FUNCTION_BLOCK LedLamp
VAR_INPUT
END_VAR
VAR_OUTPUT
END_VAR
VAR
	output AT %Q* : BOOL;
END_VAR

PROPERTY IsOff : BOOL
GET
IsOff := NOT output;
END_GET
END_PROPERTY

PROPERTY IsOn : BOOL
GET
IsOn := output;
END_GET
END_PROPERTY

METHOD Off
VAR_INPUT
END_VAR
output := FALSE;
END_METHOD

METHOD On
VAR_INPUT
END_VAR
output := TRUE;
END_METHOD

END_FUNCTION_BLOCK

(* stored: Version 1.1.0.1, ProductVersion 3.1.4024.12
   POU LedLamp: Id {3fdc688c-187e-4867-8a23-fcd2f38403ef}, SpecialFunc None
   Property IsOff: Id {3d50d815-2c1d-4f69-bd5f-d5cf14c05e56}
   Get Get: Id {a27671c2-1dca-49f2-a356-5aa69b09b24c}
   Property IsOn: Id {aec8a761-94b2-4bd0-82a2-5b083fb52d2c}
   Get Get: Id {212606ac-f0fd-42b8-9919-30c789c4546e}
   Method Off: Id {f2cced46-62eb-4e4b-bd14-f54621011151}
   Method On: Id {ab28f0e6-37ba-45ff-af1b-15e2119b2b0e} *)
